// TIA Portal V20 export
// export: Created 2026-07-16T12:58:47.0489228Z, ExportSetting WithDefaults, DisplayName Totally Integrated Automation Portal, DisplayVersion V20 Update 5, DisplayName TIA Portal Openness, DisplayVersion V20 Update 4, DisplayName TIA Portal Version Control Interface, DisplayVersion V20 Update 5, DisplayName SINAMICS Startdrive Advanced, DisplayVersion V20, DisplayName SINAMICS DCC, DisplayVersion V20, DisplayName SINAMICS Startdrive G130, G150, S120, S150, SINAMICS MV, G220, S200, S210, DisplayVersion V20, DisplayName SINAMICS Startdrive G110M, G120, G120C, G120D, G120P, G115D, DisplayVersion V20, DisplayName STEP 7 Professional, DisplayVersion V20 Update 5, DisplayName STEP 7 Safety, DisplayVersion V20 Update 2, DisplayName WinCC Basic/Comfort/Advanced, DisplayVersion V20 Update 5, DisplayName WinCC Unified, DisplayVersion V20 Update 5
DATA_BLOCK "DB_Controls"   // DB4
{ S7_Optimized_Access := 'TRUE' }
VERSION : 0.1
// Operator/HMI command surface (C-306). Written by HMI, consumed by equipment FBs and the sequencer - not logic-internal state.
// stored: AutoNumber true, DBAccessibleFromOPCUA true, IsOnlyStoredInLoadMemory false, IsRetainMemResEnabled false, IsWriteProtectedInAS false, MemoryReserve 100
   VAR
      PusherMode : Int;
      PusherManualCycleCmd : Bool;
      PusherJogExtendCmd : Bool;
      PusherJogRetractCmd : Bool;
      FaultReset : Bool;
   END_VAR
BEGIN
END_DATA_BLOCK
